(* IEC 61131-3 sources: as-opcua-enumstrings/OpcEnum/Program, 3 files *)

(* ---- Types.typ ---- *)
TYPE
	Step_typ :
		(
		STATE_WAIT, (*State_wait*)
		STATE_RUN, (*State_run*)
		STATE_STOP (*State_stop*)
		);
END_TYPE

(* ---- Main.st ---- *)
PROGRAM _INIT
	Step := STATE_WAIT;
	dStep ACCESS ADR(Step);
END_PROGRAM

PROGRAM _CYCLIC
	(* Insert code here *)

END_PROGRAM

PROGRAM _EXIT
	(* Insert code here *)

END_PROGRAM

(* ---- Variables.var ---- *)
VAR
	Step : Step_typ;
	dStep : REFERENCE TO DINT;
END_VAR
